TYPE RxMessage :
STRUCT
	length:       UINT;
	CobId:				UDINT;
	RxMessage:		ARRAY [0..7] OF USINT;
END_STRUCT
END_TYPE

(* stored: Version 1.1.0.1, ProductVersion 3.1.4022.6
   DUT RxMessage: Id {91eaedf5-f36f-4fc9-9f99-0621985e6609} *)
